{attribute 'GeneratedUsingTerminal: ELM9410-0000-0016'}
{attribute addProperty BoxType "ELM9410-0000-0016"}
{attribute addProperty Id "StatusAT %I*Status_BA3D1C5D7Number_of_samplesAT %I*UINT2"}
{attribute addProperty CRC "292982937"}
{attribute addProperty Size "9"}
TYPE MMS_Acceleration_Status_11769099 EXTENDS InputBase_8311D824 :
STRUCT
	{attribute addProperty Name "Status"}
	Status AT %I* : Status_BA3D1C5D;
	{attribute addProperty Name "Number_of_samples"}
	Number_of_samples AT %I* : UINT;
END_STRUCT
END_TYPE

(* stored: Version 1.2.0.0, ProductVersion 3.1.4024.11
   DUT MMS_Acceleration_Status_11769099: Id {099ded6f-81da-4251-b5fc-634b6ceb94b1} *)
